// TIA Portal V19 export
DATA_BLOCK "IPC_Manager"   // DB207
// stored: InstanceOfName IPC_Manager_FB, InstanceOfType FB
"IPC_Manager_FB"
   // VAR
   //    Warning : Struct
   //       Err_Send : "IPC_Msg_Send_Err";
   //    END_STRUCT;
   //    Send_Msg_Log { S7_SetPoint := 'True'} : "IPC_Send_Msg_From_Buffer_FB";
   // END_VAR
BEGIN
END_DATA_BLOCK
